FUNCTION_BLOCK Stage8 (* Template for a Basic Function Block Type *)
  (* Standard: 61499-2 *)
  (* Version 1.0, 2021-06-20, HP *)
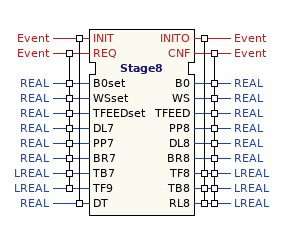
  EVENT_INPUT
    INIT WITH DT; (* Initialization Request *)
    REQ WITH B0set, WSset, TFEEDset, DL7, PP7, BR7, TB7, TF9; (* Normal Execution Request *)
  END_EVENT
  EVENT_OUTPUT
    INITO WITH TB8, RL8, TF8; (* Initialization Confirm *)
    CNF WITH TB8, DL8, TF8, TFEED, WS, PP8, BR8, RL8, B0; (* Execution Confirmation *)
  END_EVENT
  VAR_INPUT
    B0set : REAL;
    WSset : REAL;
    TFEEDset : REAL;
    DL7 : REAL;
    PP7 : REAL;
    BR7 : REAL;
    TB7 : LREAL;
    TF9 : LREAL;
    DT : REAL;
  END_VAR
  VAR_OUTPUT
    B0 : REAL;
    WS : REAL;
    TFEED : REAL;
    PP8 : REAL;
    DL8 : REAL;
    BR8 : REAL;
    TF8 : LREAL;
    TB8 : LREAL;
    RL8 : LREAL;
  END_VAR
  VAR
    AB : REAL; (* internal variabel *)
    UU : REAL;
    TREF : REAL;
    AD : REAL;
    AHC : REAL;
    AHR : REAL;
    AS : REAL;
    REC : REAL;
    WN : REAL;
    WN_1 : REAL;
    XKN : REAL;
    C1 : REAL;
    HS : REAL;
    G : REAL;
    W1 : REAL;
    TFREC : REAL;
    TS : REAL;
    DTS : REAL;
    TF8_last : REAL;
    RL8_last : REAL;
    TB8_last : REAL;
    USS : REAL;
    RHOB : REAL;
    CPB : REAL;
    CPF : REAL;
    FMW : REAL;
    HLV : REAL;
    HV : REAL;
    BPR : REAL;
    FMC : REAL;
    U : REAL;
    A : REAL;
    B : REAL;
    C : REAL;
    D1 : REAL;
    d : REAL;
    a : REAL;
    A1 : REAL;
    A2 : REAL;
    A3 : REAL;
    A4 : REAL;
    A5 : REAL;
    A6 : REAL;
    p : REAL;
    q : REAL;
    TC : REAL;
    PC : REAL;
    DTB8 : REAL;
    DEN8 : REAL;
    DH8 : REAL;
    DP8 : REAL;
    DPDH8 : REAL;
    DT8 : REAL;
    m : REAL;
    n : REAL;
    VR8 : REAL;
    DELTA8 : REAL;
    DELTA30 : REAL;
    DELTA52 : REAL;
    DELTA8_last : REAL;
    DELTA30_last : REAL;
    DELTA52_last : REAL;
  END_VAR
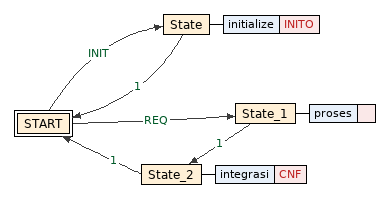
  EC_STATES
    START; (* Initial State *)
    State : initialize -> INITO;
    State_1 : proses;
    State_2 : integrasi -> CNF;
  END_STATES
  EC_TRANSITIONS
    START TO State := INIT;
    State TO START := 1;
    START TO State_1 := REQ;
    State_1 TO State_2 := 1;
    State_2 TO START := 1;
  END_TRANSITIONS
  ALGORITHM initialize IN ST: (* Initialization algorithm *)
TREF :=273.15;
AB :=57.2727;
AHC :=4069.2;
AHR :=2639.7;
AS :=3225.7;
REC :=0.0;
//TF2:=TF2;

//TFEED :=TFEED1+TREF;
 //TS:=TS1+TREF;
WN :=3.0;
XKN :=0.68;
HS:=0.11;
G :=9.81;
W1 :=0.50;

RL8 := 0.558948661515042;
TB8 := 345.783441999712;
TF8 := 341.885924485359;
TF9 := 339.272674118834;


RL8_last :=RL8;
TB8_last :=TB8;
TF8_last :=TF8;
  END_ALGORITHM
  ALGORITHM proses IN ST: (* kalkulasi *)
B0 :=B0set;
WS :=WSset;
TFEED:=TFEEDset;
UU := TFEEDset;
U :=UU;

USS :=49.767;
C1 :=0.625;
RHOB :=1032.4; //maassa jenis brine
CPB :=1.00; //heatcapacity Brine
CPF :=1.00; //heat capacity feed
FMW :=23654.0;
HLV :=563.7959;
HV :=625.1971;
BPR :=2.192;
FMC :=34736.09;
//U :=UU; //feed temp



///  Calculate the physical properties

//A :=3.2437814;
//B :=5.86826*0.001;
//C :=1.1702379*0.00000001;
//D1 :=2.1878462*0.001;
//TC :=647.27;
//PC :=218.167;


A1 :=3.2437814;
A2:=5.86826*0.001;
A3:=1.1702379*0.00000001;
A4 :=2.1878462*0.001;
A5 :=647.27;
A6 :=218.167;

DTB8 :=A5-TB8;
DEN8 :=(A1+A2*DTB8+A3*DTB8*DTB8*DTB8)/(1+A4*DTB8)*DTB8/TB8;
p:=DEN8;
q:=10.0;
PP8 :=A6/(EXPT(q, p));

// calculate the brine flow rates
DP8:=PP7-PP8;
DH8:=RL8-C1*HS;
DPDH8 :=DP8*101000+G*RHOB*DH8;
m:=DPDH8*RHOB;
n:=0.5;
BR8 :=WN*XKN*RL8*(EXPT(m, n));
BR8 :=BR8*60.0/1000.0;

// calculate the vapor flow rates

DT8 :=TB8-BPR/1.8-(TF9+TF8)*0.5;
VR8 :=U*AHC*DT8/HLV/1000.0;
DL8 :=DL7+VR8;


//// state equation
DELTA8 :=(BR7-BR8-VR8)*1000.0/RHOB/AB;
DELTA30 :=((BR7*CPB*(TB7-TB8))-VR8*(HV-CPB*(TB8-TREF)))*1000.0/AB/RHOB/CPB/RL8;
DELTA52 :=(B0*CPF*(TF9-TF8)*1000+(U*AHC*DT8))/FMW/CPF;
  END_ALGORITHM
  ALGORITHM integrasi IN ST: (* new algorithm *)
B0 :=B0set;
WS :=WSset;
TFEED:=TFEEDset;
//integrasi
RL8 := (DELTA8 + DELTA8_last)*0.5*DT + RL8_last;
DELTA8_last :=DELTA8 ;
RL8_last :=RL8;

TB8:= (DELTA30 + DELTA30_last)*0.5*DT + TB8_last;
DELTA30_last :=DELTA30 ;
TB8_last:=TB8;

TF8 := (DELTA52 + DELTA52_last)*0.5*DT + TF8_last;
DELTA52_last :=DELTA52 ;
TF8_last :=TF8;
  END_ALGORITHM
END_FUNCTION_BLOCK
